TYPE DUT_HMI_Motor_Freq EXTENDS DUT_Control_Base_Valve :
STRUCT
	ModeValue : INT:= 1; // 0: Manual; 1: Auto;
	DisableAutoManual : BOOL;
END_STRUCT
END_TYPE

(* stored: Version 1.1.0.1, ProductVersion 3.1.4024.12
   DUT DUT_HMI_Motor_Freq: Id {b5181239-9c7c-493e-8870-473dddbbad05} *)
